{region '#Template'}
	{attribute 'Version' := '5.0.0.0'}
	{attribute 'Tags' := '"LCID": "1031", "Text": "Fassade, Sonnenschutz"'}
	{attribute 'Tags' := '"LCID": "1033", "Text": "Facade, Sunprotection"'}
	{attribute 'Using' := '"Type": "Template", "URI": "ST_BA_SunBld"'}
	{attribute 'Description' := '"LCID": "1031", "Text": "Sonnenschutz Lamellennachführung"'}
	{attribute 'Description' := '"LCID": "1033", "Text": "Sunprotection slat adjustment"'}
{endregion}
FUNCTION_BLOCK FB_BA_Facade_SunProtection EXTENDS FB_BA_View
VAR_INPUT
	bFcdInSun						: BOOL;
	fFcdOrtn						: REAL;	
	fFcdAngl						: REAL;
	fLamWdth						: REAL;
	fLamDstc						: REAL;
END_VAR
VAR_OUTPUT
	stSunbld						: ST_BA_SunBld;
	bSunPrtcActv					: BOOL;
END_VAR                     
VAR_INPUT CONSTANT          
	SunPrtcValOn00deg				: FB_BA_AV_Op;	
	SunPrtcValOn15deg				: FB_BA_AV_Op;	
	SunPrtcValOn30deg				: FB_BA_AV_Op;	
	SunPrtcValOn45deg				: FB_BA_AV_Op;	
	SunPrtcValOn60deg				: FB_BA_AV_Op;	
	SunPrtcValOn75deg				: FB_BA_AV_Op;	
	SunPrtcValOn90deg				: FB_BA_AV_Op;	
				            				
	SunPrtcValOff00deg				: FB_BA_AV_Op;	
	SunPrtcValOff15deg				: FB_BA_AV_Op;	
	SunPrtcValOff30deg				: FB_BA_AV_Op;	
	SunPrtcValOff45deg				: FB_BA_AV_Op;	
	SunPrtcValOff60deg				: FB_BA_AV_Op;	
	SunPrtcValOff75deg				: FB_BA_AV_Op;	
	SunPrtcValOff90deg				: FB_BA_AV_Op;	
  
	SunPrtcValOnCalc				: FB_BA_AV_Op;				  
	SunPrtcValOffCalc				: FB_BA_AV_Op;		
	SunPrtcDlyOn					: FB_BA_AV_Op;				  
	SunPrtcDlyOff					: FB_BA_AV_Op;		
	SunPrtcState					: FB_BA_BV_Op;				  
	SunPrtcPos						: FB_BA_AV_Op;		  
	SunPrtcAngl						: FB_BA_AV_Op;		
	SunPrtc							: FB_BA_SunPrtc;	
END_VAR                     
VAR                         
	aBrtnsDirection					: ARRAY[1..32] OF REAL :=	[0.0, 90.0, 180.0, 270.0, 360.0];
	aBrtnsAtDirection				: ARRAY[1..32] OF REAL;
	
	BrtnsCardinalInterpolation		: FB_BA_Chrct32;		// brightness interpolated regarding the azimuth / Sonnenhelligkeit interpoliert nach der Sonnenrichtung
	
	SunPrtcValOn					: FB_BA_Chrct07;		// calculates the elevation-related factor for the on-values / Errechnung der sonnenhöhenabhängigen Faktoren der Einschaltschwelle	
	SunPrtcValOff					: FB_BA_Chrct07;		// calculates the elevation-related factor for the off-values / Errechnung der sonnenhöhenabhängigen Faktoren der Ausschaltschwelle	

	SunPrtcValOnOff					: FB_BA_Swi2P;
END_VAR

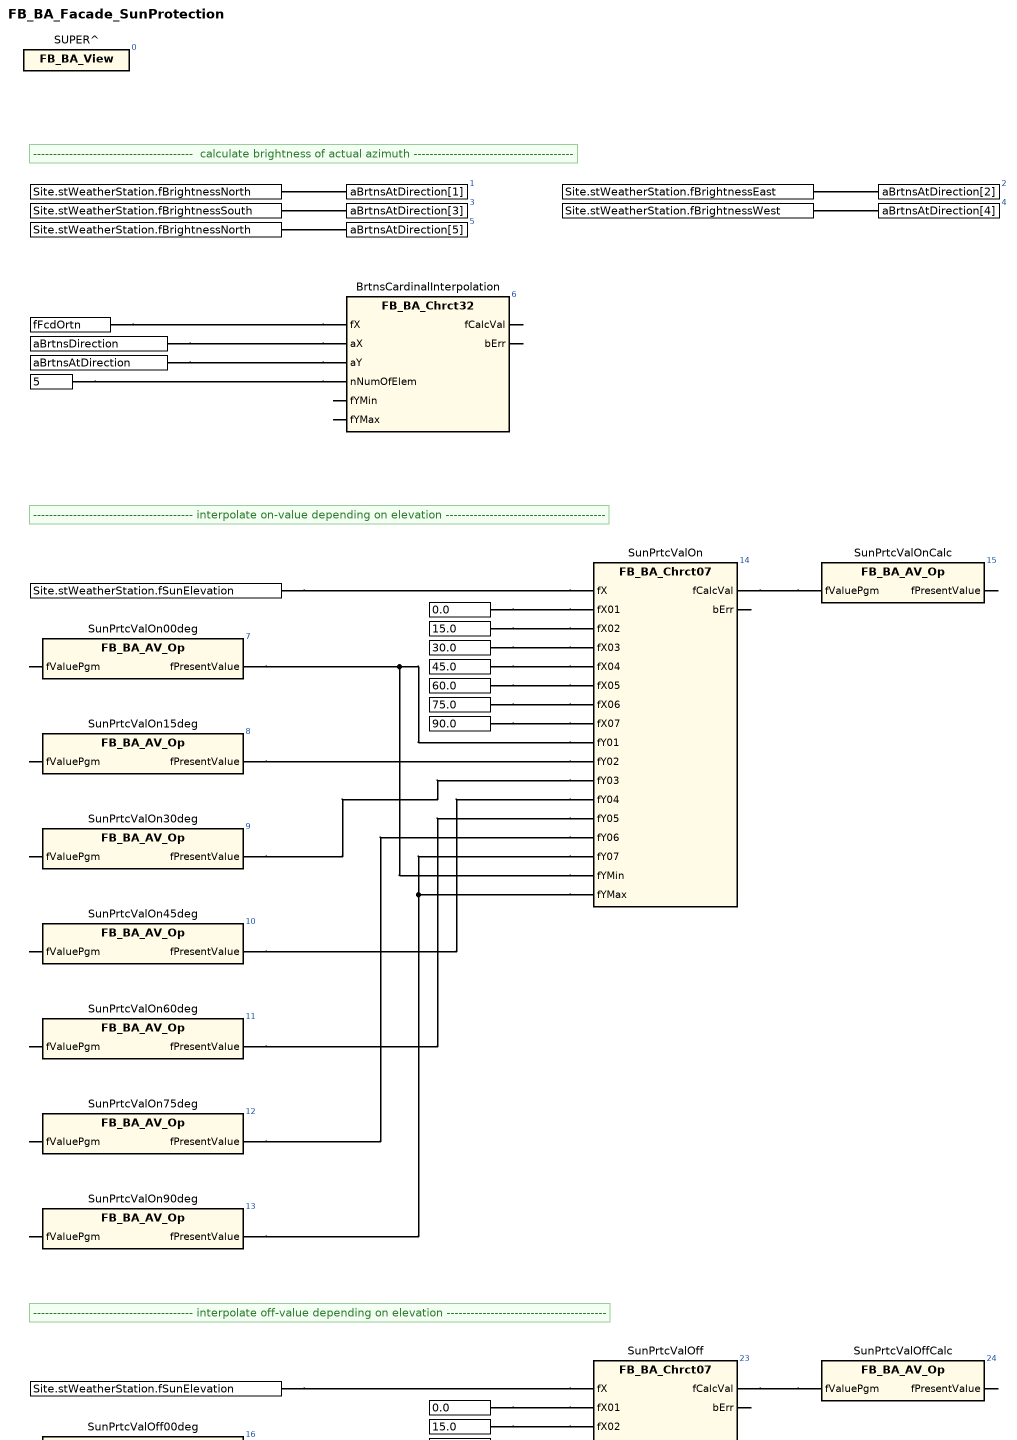
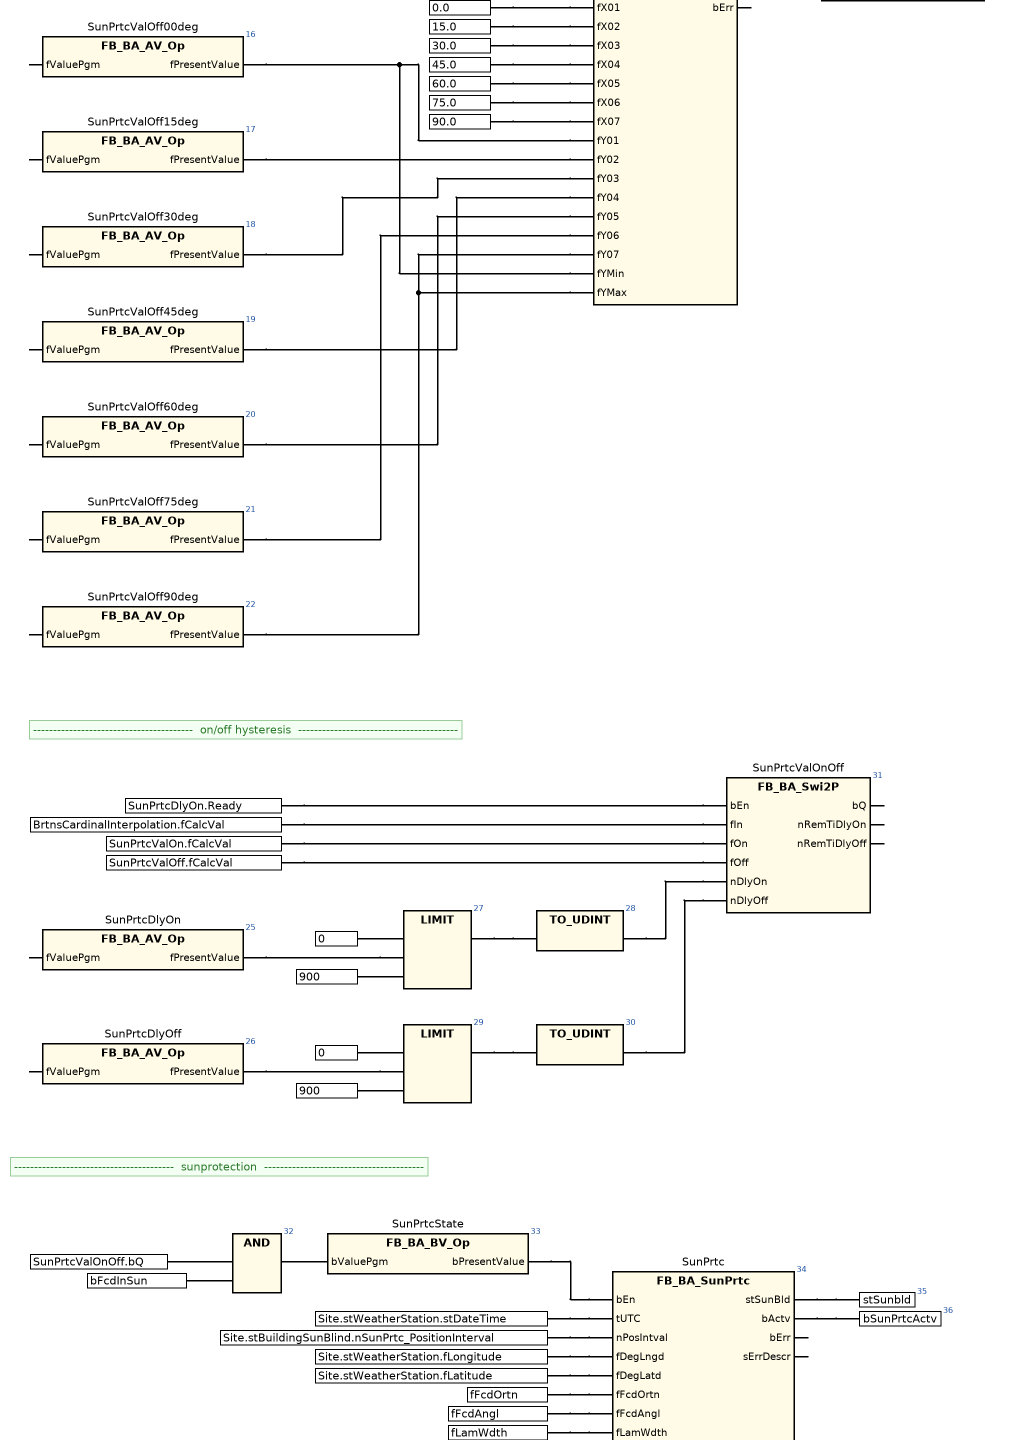
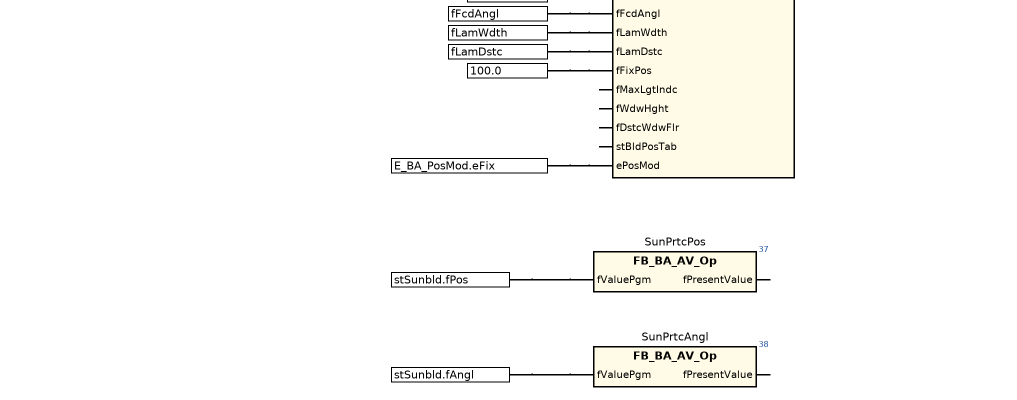
SUPER^(); // FB_BA_View
// ----------------------------------------  calculate brightness of actual azimuth ----------------------------------------
aBrtnsAtDirection[1] := Site.stWeatherStation.fBrightnessNorth;
aBrtnsAtDirection[2] := Site.stWeatherStation.fBrightnessEast;
aBrtnsAtDirection[3] := Site.stWeatherStation.fBrightnessSouth;
aBrtnsAtDirection[4] := Site.stWeatherStation.fBrightnessWest;
aBrtnsAtDirection[5] := Site.stWeatherStation.fBrightnessNorth;
BrtnsCardinalInterpolation(fX := fFcdOrtn, aX := aBrtnsDirection, aY := aBrtnsAtDirection, nNumOfElem := 5); // FB_BA_Chrct32
// ---------------------------------------- interpolate on-value depending on elevation ----------------------------------------
SunPrtcValOn00deg(); // FB_BA_AV_Op
SunPrtcValOn15deg(); // FB_BA_AV_Op
SunPrtcValOn30deg(); // FB_BA_AV_Op
SunPrtcValOn45deg(); // FB_BA_AV_Op
SunPrtcValOn60deg(); // FB_BA_AV_Op
SunPrtcValOn75deg(); // FB_BA_AV_Op
SunPrtcValOn90deg(); // FB_BA_AV_Op
SunPrtcValOn(
    fX := Site.stWeatherStation.fSunElevation,
    fX01 := 0.0,
    fX02 := 15.0,
    fX03 := 30.0,
    fX04 := 45.0,
    fX05 := 60.0,
    fX06 := 75.0,
    fX07 := 90.0,
    fY01 := SunPrtcValOn00deg.fPresentValue,
    fY02 := SunPrtcValOn15deg.fPresentValue,
    fY03 := SunPrtcValOn30deg.fPresentValue,
    fY04 := SunPrtcValOn45deg.fPresentValue,
    fY05 := SunPrtcValOn60deg.fPresentValue,
    fY06 := SunPrtcValOn75deg.fPresentValue,
    fY07 := SunPrtcValOn90deg.fPresentValue,
    fYMin := SunPrtcValOn00deg.fPresentValue,
    fYMax := SunPrtcValOn90deg.fPresentValue); // FB_BA_Chrct07
SunPrtcValOnCalc(fValuePgm := SunPrtcValOn.fCalcVal); // FB_BA_AV_Op
// ---------------------------------------- interpolate off-value depending on elevation ----------------------------------------
SunPrtcValOff00deg(); // FB_BA_AV_Op
SunPrtcValOff15deg(); // FB_BA_AV_Op
SunPrtcValOff30deg(); // FB_BA_AV_Op
SunPrtcValOff45deg(); // FB_BA_AV_Op
SunPrtcValOff60deg(); // FB_BA_AV_Op
SunPrtcValOff75deg(); // FB_BA_AV_Op
SunPrtcValOff90deg(); // FB_BA_AV_Op
SunPrtcValOff(
    fX := Site.stWeatherStation.fSunElevation,
    fX01 := 0.0,
    fX02 := 15.0,
    fX03 := 30.0,
    fX04 := 45.0,
    fX05 := 60.0,
    fX06 := 75.0,
    fX07 := 90.0,
    fY01 := SunPrtcValOff00deg.fPresentValue,
    fY02 := SunPrtcValOff15deg.fPresentValue,
    fY03 := SunPrtcValOff30deg.fPresentValue,
    fY04 := SunPrtcValOff45deg.fPresentValue,
    fY05 := SunPrtcValOff60deg.fPresentValue,
    fY06 := SunPrtcValOff75deg.fPresentValue,
    fY07 := SunPrtcValOff90deg.fPresentValue,
    fYMin := SunPrtcValOff00deg.fPresentValue,
    fYMax := SunPrtcValOff90deg.fPresentValue); // FB_BA_Chrct07
SunPrtcValOffCalc(fValuePgm := SunPrtcValOff.fCalcVal); // FB_BA_AV_Op
// ----------------------------------------  on/off hysteresis  ----------------------------------------
SunPrtcDlyOn(); // FB_BA_AV_Op
SunPrtcDlyOff(); // FB_BA_AV_Op
SunPrtcValOnOff(
    bEn := SunPrtcDlyOn.Ready,
    fIn := BrtnsCardinalInterpolation.fCalcVal,
    fOn := SunPrtcValOn.fCalcVal,
    fOff := SunPrtcValOff.fCalcVal,
    nDlyOn := TO_UDINT(LIMIT(0, SunPrtcDlyOn.fPresentValue, 900)),
    nDlyOff := TO_UDINT(LIMIT(0, SunPrtcDlyOff.fPresentValue, 900))); // FB_BA_Swi2P
// ----------------------------------------  sunprotection  ----------------------------------------
SunPrtcState(bValuePgm := SunPrtcValOnOff.bQ AND bFcdInSun); // FB_BA_BV_Op
SunPrtc(
    bEn := SunPrtcState.bPresentValue,
    tUTC := Site.stWeatherStation.stDateTime,
    nPosIntval := Site.stBuildingSunBlind.nSunPrtc_PositionInterval,
    fDegLngd := Site.stWeatherStation.fLongitude,
    fDegLatd := Site.stWeatherStation.fLatitude,
    fFcdOrtn := fFcdOrtn,
    fFcdAngl := fFcdAngl,
    fLamWdth := fLamWdth,
    fLamDstc := fLamDstc,
    fFixPos := 100.0,
    ePosMod := E_BA_PosMod.eFix); // FB_BA_SunPrtc
stSunbld := SunPrtc.stSunBld;
bSunPrtcActv := SunPrtc.bActv;
SunPrtcPos(fValuePgm := stSunbld.fPos); // FB_BA_AV_Op
SunPrtcAngl(fValuePgm := stSunbld.fAngl); // FB_BA_AV_Op

METHOD FB_init : BOOL
VAR_INPUT
	bInitRetains : BOOL; // if TRUE; the retain variables are initialized (warm start / cold start)
	bInCopyCode : BOOL;  // if TRUE; the instance afterwards gets moved into the copy code (online change)
END_VAR
SunPrtcValOn00deg.iParent		:= THIS^;
SunPrtcValOn00deg.iLabel		:= LblCtl_SunProtectionValueOn0deg;
SunPrtcValOn00deg.eUnit			:= E_BA_Unit.eOther_NoUnits; 
SunPrtcValOn00deg.fValueRm		:= 3000;

SunPrtcValOn15deg.iParent		:= THIS^;
SunPrtcValOn15deg.iLabel		:= LblCtl_SunProtectionValueOn15deg;
SunPrtcValOn15deg.eUnit			:= E_BA_Unit.eOther_NoUnits; 
SunPrtcValOn15deg.fValueRm		:= 10000;

SunPrtcValOn30deg.iParent		:= THIS^;
SunPrtcValOn30deg.iLabel		:= LblCtl_SunProtectionValueOn30deg;
SunPrtcValOn30deg.eUnit			:= E_BA_Unit.eOther_NoUnits; 
SunPrtcValOn30deg.fValueRm		:= 40000;
	
SunPrtcValOn45deg.iParent		:= THIS^;
SunPrtcValOn45deg.iLabel		:= LblCtl_SunProtectionValueOn45deg;
SunPrtcValOn45deg.eUnit			:= E_BA_Unit.eOther_NoUnits; 
SunPrtcValOn45deg.fValueRm		:= 80000;

SunPrtcValOn60deg.iParent		:= THIS^;
SunPrtcValOn60deg.iLabel		:= LblCtl_SunProtectionValueOn60deg;
SunPrtcValOn60deg.eUnit			:= E_BA_Unit.eOther_NoUnits; 
SunPrtcValOn60deg.fValueRm		:= 120000;

SunPrtcValOn75deg.iParent		:= THIS^;
SunPrtcValOn75deg.iLabel		:= LblCtl_SunProtectionValueOn75deg;
SunPrtcValOn75deg.eUnit			:= E_BA_Unit.eOther_NoUnits; 
SunPrtcValOn75deg.fValueRm		:= 160000;

SunPrtcValOn90deg.iParent		:= THIS^;
SunPrtcValOn90deg.iLabel		:= LblCtl_SunProtectionValueOn90deg;
SunPrtcValOn90deg.eUnit			:= E_BA_Unit.eOther_NoUnits; 
SunPrtcValOn90deg.fValueRm		:= 200000;


SunPrtcValOff00deg.iParent		:= THIS^;
SunPrtcValOff00deg.iLabel		:= LblCtl_SunProtectionValueOff0deg;
SunPrtcValOff00deg.eUnit		:= E_BA_Unit.eOther_NoUnits; 
SunPrtcValOff00deg.fValueRm		:= 1000;
                  
SunPrtcValOff15deg.iParent		:= THIS^;
SunPrtcValOff15deg.iLabel		:= LblCtl_SunProtectionValueOff15deg;
SunPrtcValOff15deg.eUnit		:= E_BA_Unit.eOther_NoUnits; 
SunPrtcValOff15deg.fValueRm		:= 8000;
                  
SunPrtcValOff30deg.iParent		:= THIS^;
SunPrtcValOff30deg.iLabel		:= LblCtl_SunProtectionValueOff30deg;
SunPrtcValOff30deg.eUnit		:= E_BA_Unit.eOther_NoUnits; 
SunPrtcValOff30deg.fValueRm		:= 30000;
                  
SunPrtcValOff45deg.iParent		:= THIS^;
SunPrtcValOff45deg.iLabel		:= LblCtl_SunProtectionValueOff45deg;
SunPrtcValOff45deg.eUnit		:= E_BA_Unit.eOther_NoUnits; 
SunPrtcValOff45deg.fValueRm		:= 60000;
                  
SunPrtcValOff60deg.iParent		:= THIS^;
SunPrtcValOff60deg.iLabel		:= LblCtl_SunProtectionValueOff60deg;
SunPrtcValOff60deg.eUnit		:= E_BA_Unit.eOther_NoUnits; 
SunPrtcValOff60deg.fValueRm		:= 90000;
                  
SunPrtcValOff75deg.iParent		:= THIS^;
SunPrtcValOff75deg.iLabel		:= LblCtl_SunProtectionValueOff75deg;
SunPrtcValOff75deg.eUnit		:= E_BA_Unit.eOther_NoUnits; 
SunPrtcValOff75deg.fValueRm		:= 120000;
                  
SunPrtcValOff90deg.iParent		:= THIS^;
SunPrtcValOff90deg.iLabel		:= LblCtl_SunProtectionValueOff90deg;
SunPrtcValOff90deg.eUnit		:= E_BA_Unit.eOther_NoUnits; 
SunPrtcValOff90deg.fValueRm		:= 150000;



SunPrtcValOnCalc.iParent		:= THIS^;
SunPrtcValOnCalc.iLabel			:= LblCtl_SunProtectionValueOnCalc;
SunPrtcValOnCalc.eUnit			:= E_BA_Unit.eLight_Luxes; 
                                							    
SunPrtcValOffCalc.iParent		:= THIS^;
SunPrtcValOffCalc.iLabel		:= LblCtl_SunProtectionValueOffCalc;
SunPrtcValOffCalc.eUnit			:= E_BA_Unit.eLight_Luxes; 
                                
SunPrtcDlyOn.iParent			:= THIS^;
SunPrtcDlyOn.iLabel				:= LblCtl_TimeDelaySunProtectionOn;
SunPrtcDlyOn.eUnit				:= E_BA_Unit.eTime_Seconds; 
SunPrtcDlyOn.fValueRm			:= 300.0;
							    
SunPrtcDlyOff.iParent			:= THIS^;
SunPrtcDlyOff.iLabel			:= LblCtl_TimeDelaySunProtectionOff;
SunPrtcDlyOff.eUnit				:= E_BA_Unit.eTime_Seconds; 
SunPrtcDlyOff.fValueRm			:= 500.0;
                                
SunPrtcState.iParent			:= THIS^;	
SunPrtcState.iLabel				:= LblCtl_SunProtectionState;
SunPrtcState.sInactiveText		:= txtEvent_Off;
SunPrtcState.sActiveText		:= txtEvent_On;
SunPrtcState.bValueRm			:= FALSE;								
SunPrtcState.eToggleMode 		:= E_BA_ToggleMode.eSwitch;	
                                
SunPrtcPos.iParent				:= THIS^;
SunPrtcPos.iLabel				:= LblFun_SunPrtcPosition;
SunPrtcPos.eUnit				:= E_BA_Unit.eTime_Seconds; 
SunPrtcPos.fValueRm				:= 300.0;
							    
SunPrtcAngl.iParent				:= THIS^;
SunPrtcAngl.iLabel				:= LblFun_SunPrtcAngle;
SunPrtcAngl.eUnit				:= E_BA_Unit.eTime_Seconds; 
SunPrtcAngl.fValueRm			:= 500.0;
END_METHOD

END_FUNCTION_BLOCK

(* stored: Version 1.1.0.1, ProductVersion 3.1.4024.12
   POU FB_BA_Facade_SunProtection: Id {3509d9b9-08c1-4ab3-9cb8-d930fa551393}, SpecialFunc None
   Method FB_init: Id {5c0b7509-a6ef-4483-be2e-557add2b86d8} *)
